// Core §8.13 — the site convention changes configuration, not mapping code.
TYPE ST_SignalTowerParCfg :
STRUCT
    SchemaVersion     : UINT := 1;
    LampTestDuration  : TIME := T#3S;
    OperatorUsesWhite : BOOL;
    HornOnHigh        : BOOL := TRUE;
END_STRUCT
END_TYPE

(* stored: Version 1.1.0.1, ProductVersion 3.1.4024.12
   DUT ST_SignalTowerParCfg: Id {f092de28-0eb8-4527-af25-d85be5ead153} *)
